(* Logix 5000 project; controller Amvex_Thorpe_Flowmeter vendor 1 type 14 code 106 rev 33.13; software revision 33.01; part 2 of 16 *)
(* tags used below, declared in another part *)
   Close : BOOL;
   Delay : TIMER;
   Open : BOOL;

ADD_ON_INSTRUCTION Banner_XS26_RCD_Function   (* revision 1.1, vendor Banner Engineering *)
// This AOI goes through a Virtual Reset or Cancel Delay request from the PLC to the XS26 Safety Controller.
VAR_IN_OUT
   RCD_Desired_Code : INT; {required}   // Numerical code that will be sent to the XS26 controller.
   RCD_Actuation_Code : INT; {required}   // Location of Actuation Code in the XS26 Controller.
   RCD_Actuation_Code_Feedback : INT; {required}   // When the Reset or Cancel Delay is successfull the Actuation Code is stored into this location.
   RCD_Bit : BOOL; {required}   // Bit that activates a singular Reset or Cancel Delay function.
   RCD_Bit_Feedback : BOOL; {required}   // Feedback bit from the XS26 controller for the RCD_Bit.
   Reset_Control_Bit : BOOL; {required}   // Bit that is turned off after the AOI completes.
   Routine_Error : BOOL; {required}
END_VAR
VAR
   Routine_Control_Bit : SINT; {access None}   // Controls operation of the AOI.
   Timer : TIMER := (PRE := 3000); {access None}
   Halt : DINT; {access None}
END_VAR

ROUTINE Logic   (* ladder *)
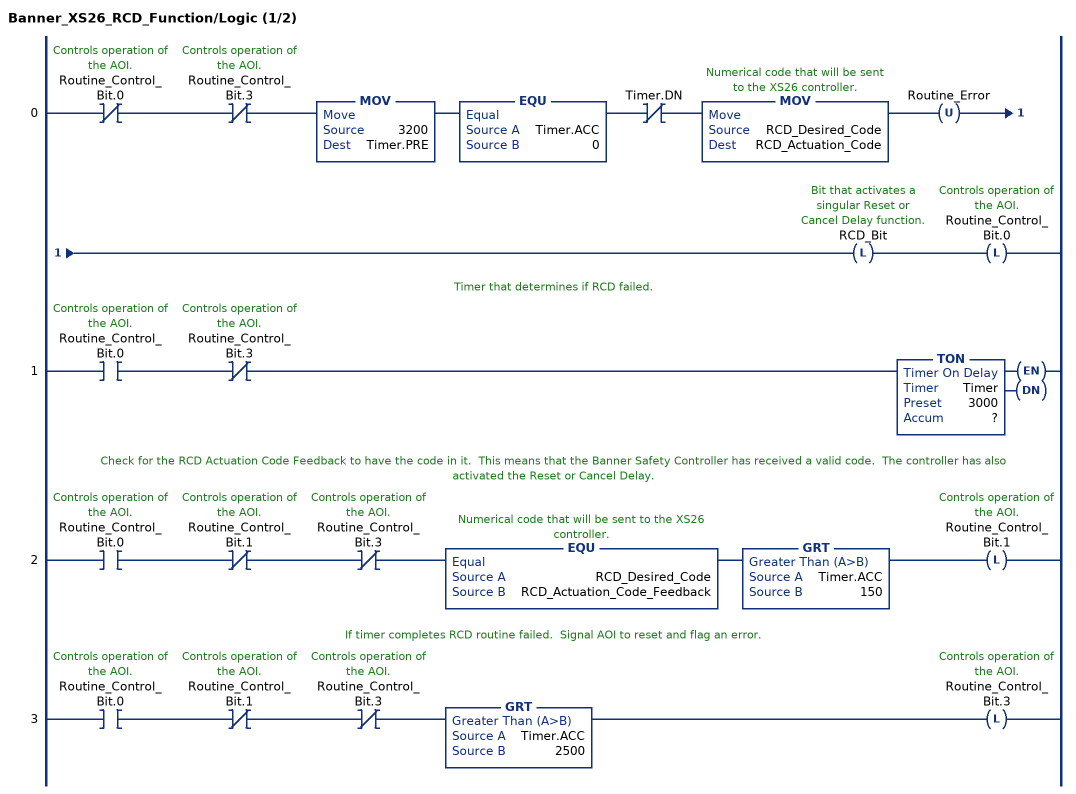
   0: XIO(Routine_Control_Bit.0)XIO(Routine_Control_Bit.3)MOV(3200,Timer.PRE)EQU(Timer.ACC,0)XIO(Timer.DN)MOV(RCD_Desired_Code,RCD_Actuation_Code)OTU(Routine_Error)OTL(RCD_Bit)OTL(Routine_Control_Bit.0);
   // Timer that determines if RCD failed.
   1: XIC(Routine_Control_Bit.0)XIO(Routine_Control_Bit.3)TON(Timer,?,?);
   // Check for the RCD Actuation Code Feedback to have the code in it.  This means that the Banner Safety Controller has received a valid code.  The controller has also activated the Reset or Cancel Delay.
   2: XIC(Routine_Control_Bit.0)XIO(Routine_Control_Bit.1)XIO(Routine_Control_Bit.3)EQU(RCD_Desired_Code,RCD_Actuation_Code_Feedback)GRT(Timer.ACC,150)OTL(Routine_Control_Bit.1);
   // If timer completes RCD routine failed.  Signal AOI to reset and flag an error.
   3: XIC(Routine_Control_Bit.0)XIO(Routine_Control_Bit.1)XIO(Routine_Control_Bit.3)GRT(Timer.ACC,2500)OTL(Routine_Control_Bit.3);
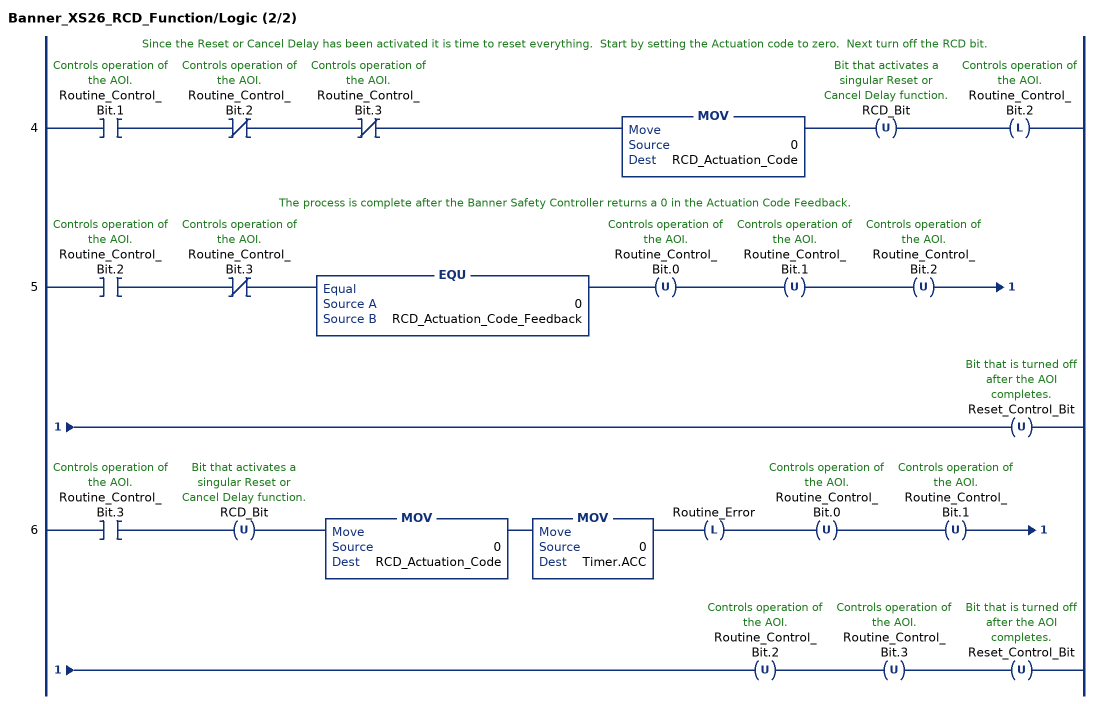
   // Since the Reset or Cancel Delay has been activated it is time to reset everything.  Start by setting the Actuation code to zero.  Next turn off the RCD bit.
   4: XIC(Routine_Control_Bit.1)XIO(Routine_Control_Bit.2)XIO(Routine_Control_Bit.3)MOV(0,RCD_Actuation_Code)OTU(RCD_Bit)OTL(Routine_Control_Bit.2);
   // The process is complete after the Banner Safety Controller returns a 0 in the Actuation Code Feedback.
   5: XIC(Routine_Control_Bit.2)XIO(Routine_Control_Bit.3)EQU(0,RCD_Actuation_Code_Feedback)OTU(Routine_Control_Bit.0)OTU(Routine_Control_Bit.1)OTU(Routine_Control_Bit.2)OTU(Reset_Control_Bit);
   6: XIC(Routine_Control_Bit.3)OTU(RCD_Bit)MOV(0,RCD_Actuation_Code)MOV(0,Timer.ACC)OTL(Routine_Error)OTU(Routine_Control_Bit.0)OTU(Routine_Control_Bit.1)OTU(Routine_Control_Bit.2)OTU(Routine_Control_Bit.3)OTU(Reset_Control_Bit);
END_ROUTINE
END_ADD_ON_INSTRUCTION

ADD_ON_INSTRUCTION Connect   (* revision 0.1, vendor Mecademic Inc. *)
// Monitor the robot module connection
VAR_IN_OUT
   RobotInstance : MODULE; {required}
END_VAR
VAR_INPUT
   Connect : BOOL; {access None, required}
END_VAR
VAR_OUTPUT
   RobotConnected : BOOL; {visible}
   ConnectionInhibited : BOOL; {visible}
   ConnectionFailed : BOOL; {visible}
END_VAR
VAR
   ConnectValue : DINT; {access None}
   DisconnectValue : DINT := 4; {access None}
   RobotInstance_Status : DINT; {access None}
   RobotInstance_Status_Masked : DINT; {access None}
END_VAR

ROUTINE Logic   (* ladder *)
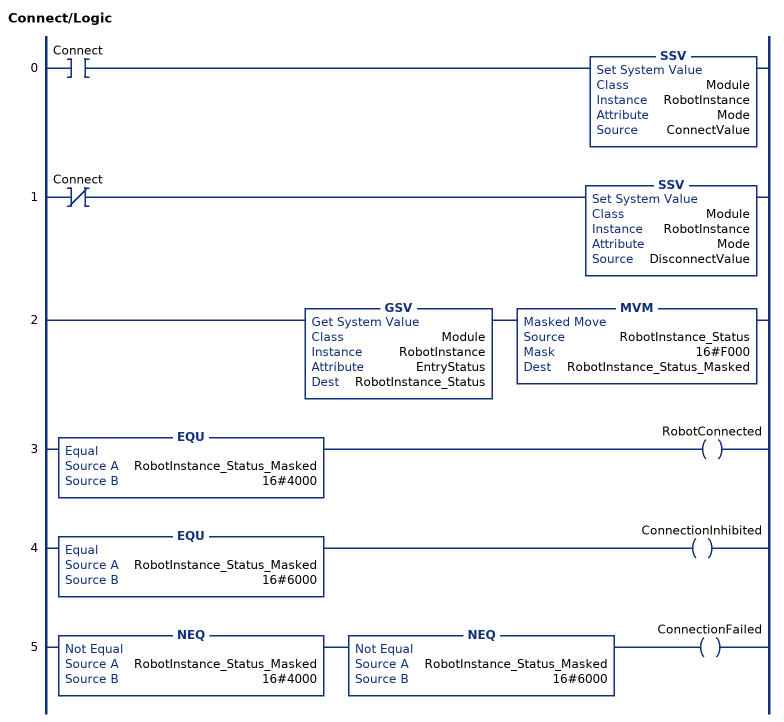
   0: XIC(Connect)SSV(Module,RobotInstance,Mode,ConnectValue);
   1: XIO(Connect)SSV(Module,RobotInstance,Mode,DisconnectValue);
   2: GSV(Module,RobotInstance,EntryStatus,RobotInstance_Status)MVM(RobotInstance_Status,16#F000,RobotInstance_Status_Masked);
   3: EQU(RobotInstance_Status_Masked,16#4000)OTE(RobotConnected);
   4: EQU(RobotInstance_Status_Masked,16#6000)OTE(ConnectionInhibited);
   5: NEQ(RobotInstance_Status_Masked,16#4000)NEQ(RobotInstance_Status_Masked,16#6000)OTE(ConnectionFailed);
END_ROUTINE
END_ADD_ON_INSTRUCTION

ADD_ON_INSTRUCTION Delay   (* revision 0.1, vendor Mecademic Inc., ExecuteEnableInFalse *)
// Delay in seconds before processing the next command
VAR_IN_OUT
   RobotInputs : _061D:Meca500_86BDA20B:I:0; {required}
   RobotOutputs : _061D:Meca500_01F88326:O:0; {required}
END_VAR
VAR_INPUT
   Parameter_Value : REAL; {required}
   ExternalStateControl : BOOL; {required}
   ExternalMoveID : INT; {required}
END_VAR
VAR_OUTPUT
   Enabled : BOOL; {visible}
   Sent : BOOL; {visible}
   Buffered : BOOL; {visible}
   Error : BOOL; {visible}
END_VAR
VAR
   InternalMoveID : INT; {access None}
   MoveIDTrig : BOOL; {access None}
   MoveIDUpdated : BOOL; {access None}
   OneShot : DINT; {access None}
   FirstScan : BOOL; {access None}
END_VAR

ROUTINE EnableInFalse   (* ladder *)
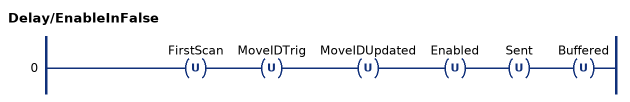
   0: OTU(FirstScan)OTU(MoveIDTrig)OTU(MoveIDUpdated)OTU(Enabled)OTU(Sent)OTU(Buffered);
END_ROUTINE

ROUTINE Logic   (* ladder *)
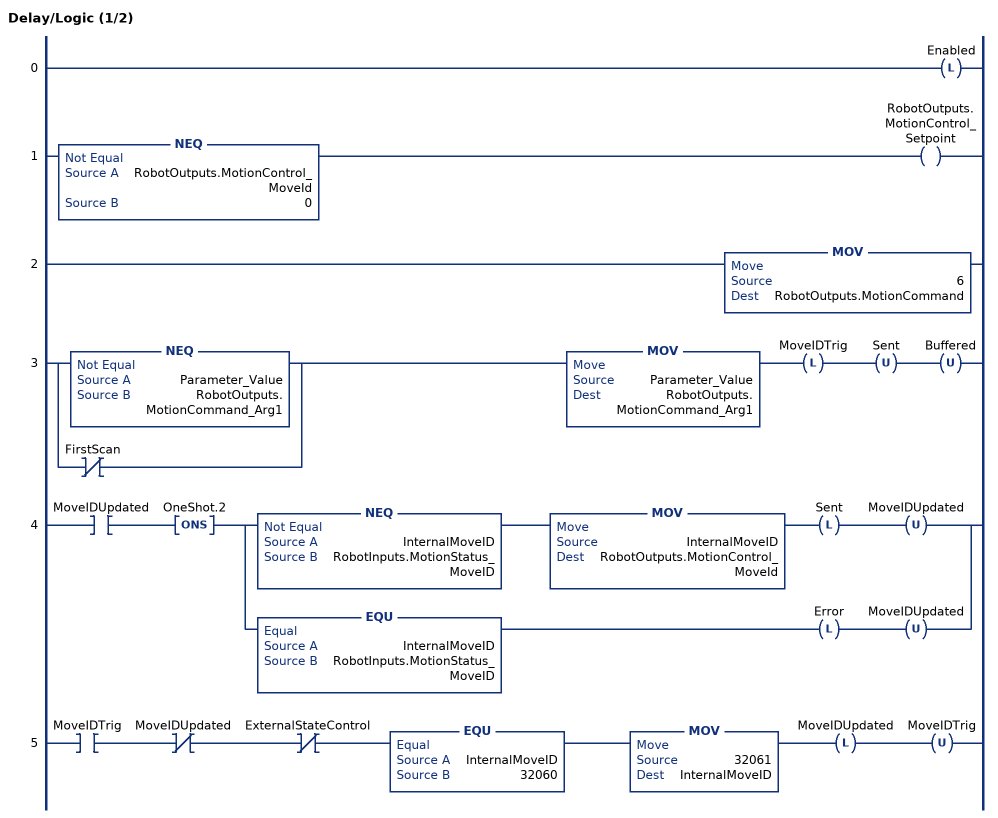
   0: OTL(Enabled);
   1: NEQ(RobotOutputs.MotionControl_MoveId,0)OTE(RobotOutputs.MotionControl_Setpoint);
   2: MOV(6,RobotOutputs.MotionCommand);
   3: [NEQ(Parameter_Value,RobotOutputs.MotionCommand_Arg1) ,XIO(FirstScan) ]MOV(Parameter_Value,RobotOutputs.MotionCommand_Arg1)OTL(MoveIDTrig)OTU(Sent)OTU(Buffered);
   4: XIC(MoveIDUpdated)ONS(OneShot.2)[NEQ(InternalMoveID,RobotInputs.MotionStatus_MoveID) MOV(InternalMoveID,RobotOutputs.MotionControl_MoveId) OTL(Sent) OTU(MoveIDUpdated) ,EQU(InternalMoveID,RobotInputs.MotionStatus_MoveID) OTL(Error) OTU(MoveIDUpdated) ];
   5: XIC(MoveIDTrig)XIO(MoveIDUpdated)XIO(ExternalStateControl)EQU(InternalMoveID,32060)MOV(32061,InternalMoveID)OTL(MoveIDUpdated)OTU(MoveIDTrig);
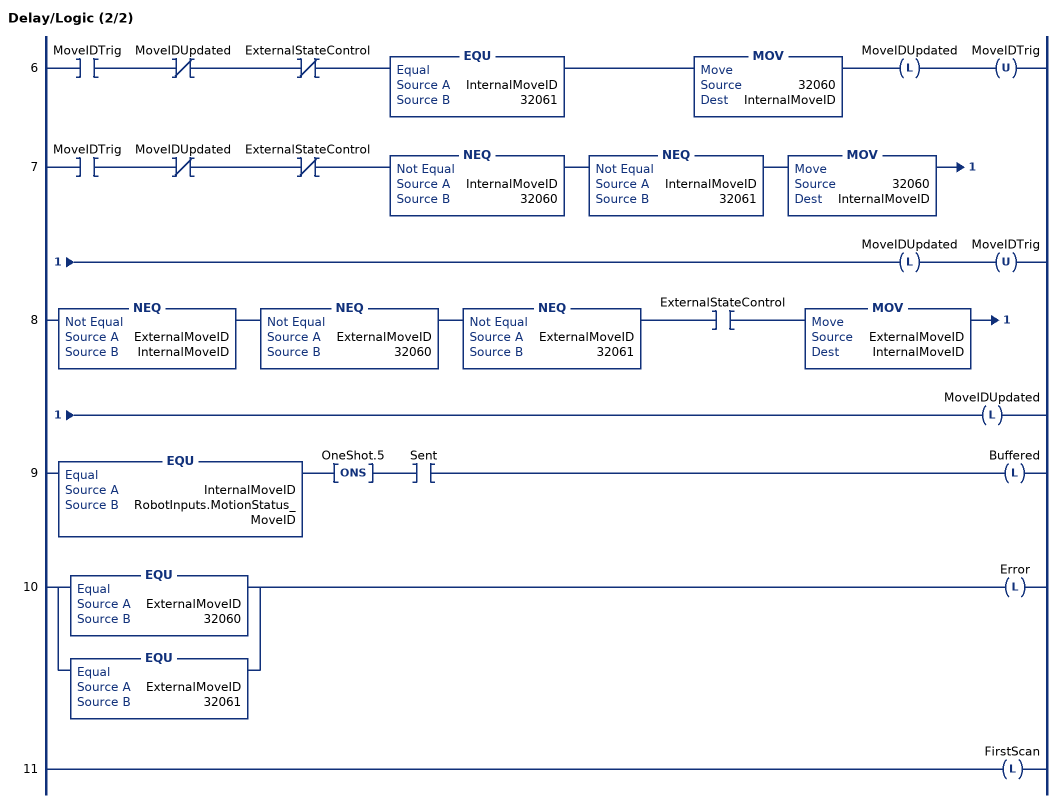
   6: XIC(MoveIDTrig)XIO(MoveIDUpdated)XIO(ExternalStateControl)EQU(InternalMoveID,32061)MOV(32060,InternalMoveID)OTL(MoveIDUpdated)OTU(MoveIDTrig);
   7: XIC(MoveIDTrig)XIO(MoveIDUpdated)XIO(ExternalStateControl)NEQ(InternalMoveID,32060)NEQ(InternalMoveID,32061)MOV(32060,InternalMoveID)OTL(MoveIDUpdated)OTU(MoveIDTrig);
   8: NEQ(ExternalMoveID,InternalMoveID)NEQ(ExternalMoveID,32060)NEQ(ExternalMoveID,32061)XIC(ExternalStateControl)MOV(ExternalMoveID,InternalMoveID)OTL(MoveIDUpdated);
   9: EQU(InternalMoveID,RobotInputs.MotionStatus_MoveID)ONS(OneShot.5)XIC(Sent)OTL(Buffered);
   10: [EQU(ExternalMoveID,32060) ,EQU(ExternalMoveID,32061) ]OTL(Error);
   11: OTL(FirstScan);
END_ROUTINE
END_ADD_ON_INSTRUCTION

ADD_ON_INSTRUCTION FAULT_AOI   (* revision 1.0, vendor Envision Automation & Controls *)
VAR_INPUT
   Fault : BOOL; {required}
   Bypass : BOOL; {required}
   Timer_PRE : DINT; {required}
END_VAR
VAR_OUTPUT
   Timer_ACC : DINT; {visible}
   Faulted : BOOL; {access Read Only, required}
END_VAR
VAR_INPUT
   Reset : BOOL; {access Read Only, required}
END_VAR
VAR
   Timer : TIMER; {access None}
END_VAR

ROUTINE Logic   (* ladder *)
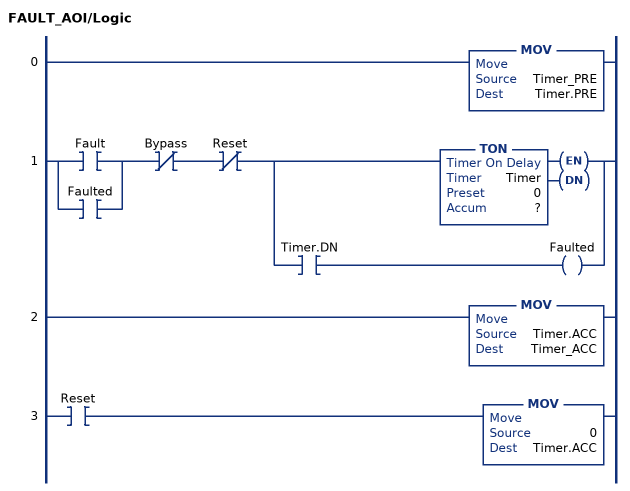
   0: MOV(Timer_PRE,Timer.PRE);
   1: [XIC(Fault) ,XIC(Faulted) ]XIO(Bypass)XIO(Reset)[TON(Timer,?,?) ,XIC(Timer.DN) OTE(Faulted) ];
   2: MOV(Timer.ACC,Timer_ACC);
   3: XIC(Reset)MOV(0,Timer.ACC);
END_ROUTINE
END_ADD_ON_INSTRUCTION

ADD_ON_INSTRUCTION GripperControl   (* revision 0.1, vendor Mecademic Inc., ExecuteEnableInFalse *)
// Open or close the gripper
VAR_IN_OUT
   RobotInputs : _061D:Meca500_86BDA20B:I:0; {required}
   RobotOutputs : _061D:Meca500_01F88326:O:0; {required}
END_VAR
VAR_INPUT
   Parameter_Value : REAL; {required}
   ExternalStateControl : BOOL; {required}
   ExternalMoveID : INT; {required}
END_VAR
VAR_OUTPUT
   Enabled : BOOL; {visible}
   Sent : BOOL; {visible}
   Buffered : BOOL; {visible}
   Error : BOOL; {visible}
END_VAR
VAR
   InternalMoveID : INT; {access None}
   MoveIDTrig : BOOL; {access None}
   MoveIDUpdated : BOOL; {access None}
   OneShot : DINT; {access None}
   FirstScan : BOOL; {access None}
END_VAR

ROUTINE EnableInFalse   (* ladder *)
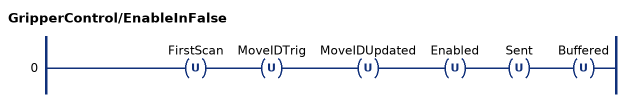
   0: OTU(FirstScan)OTU(MoveIDTrig)OTU(MoveIDUpdated)OTU(Enabled)OTU(Sent)OTU(Buffered);
END_ROUTINE

ROUTINE Logic   (* ladder *)
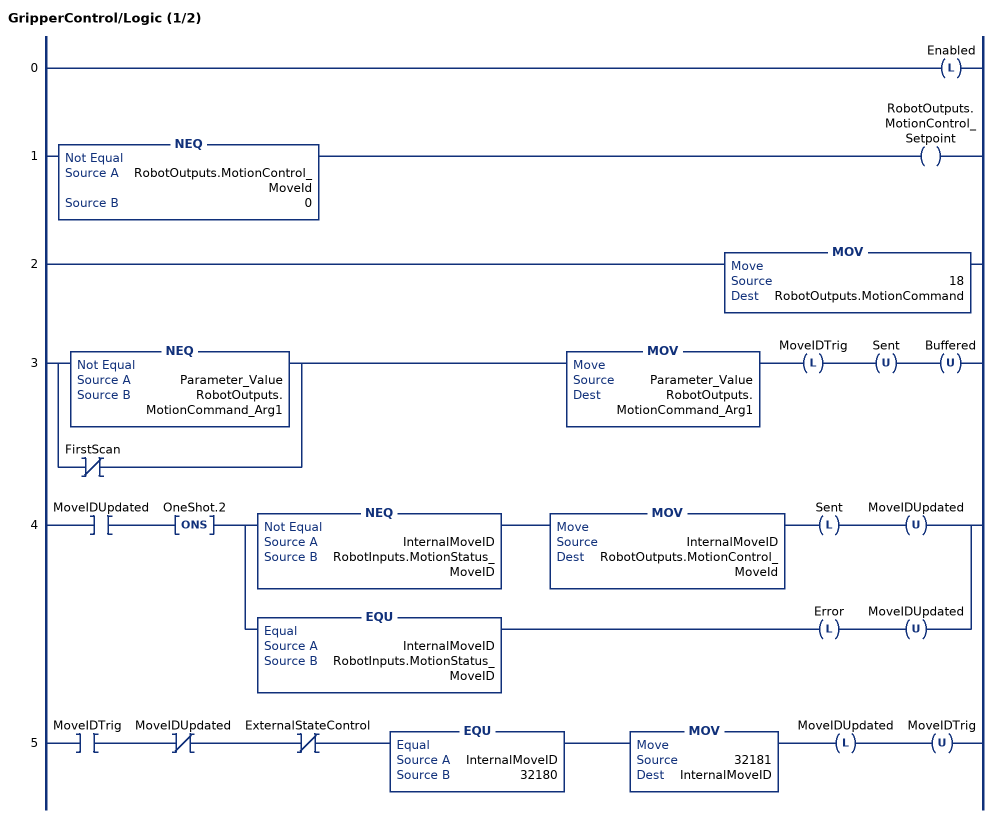
   0: OTL(Enabled);
   1: NEQ(RobotOutputs.MotionControl_MoveId,0)OTE(RobotOutputs.MotionControl_Setpoint);
   2: MOV(18,RobotOutputs.MotionCommand);
   3: [NEQ(Parameter_Value,RobotOutputs.MotionCommand_Arg1) ,XIO(FirstScan) ]MOV(Parameter_Value,RobotOutputs.MotionCommand_Arg1)OTL(MoveIDTrig)OTU(Sent)OTU(Buffered);
   4: XIC(MoveIDUpdated)ONS(OneShot.2)[NEQ(InternalMoveID,RobotInputs.MotionStatus_MoveID) MOV(InternalMoveID,RobotOutputs.MotionControl_MoveId) OTL(Sent) OTU(MoveIDUpdated) ,EQU(InternalMoveID,RobotInputs.MotionStatus_MoveID) OTL(Error) OTU(MoveIDUpdated) ];
   5: XIC(MoveIDTrig)XIO(MoveIDUpdated)XIO(ExternalStateControl)EQU(InternalMoveID,32180)MOV(32181,InternalMoveID)OTL(MoveIDUpdated)OTU(MoveIDTrig);
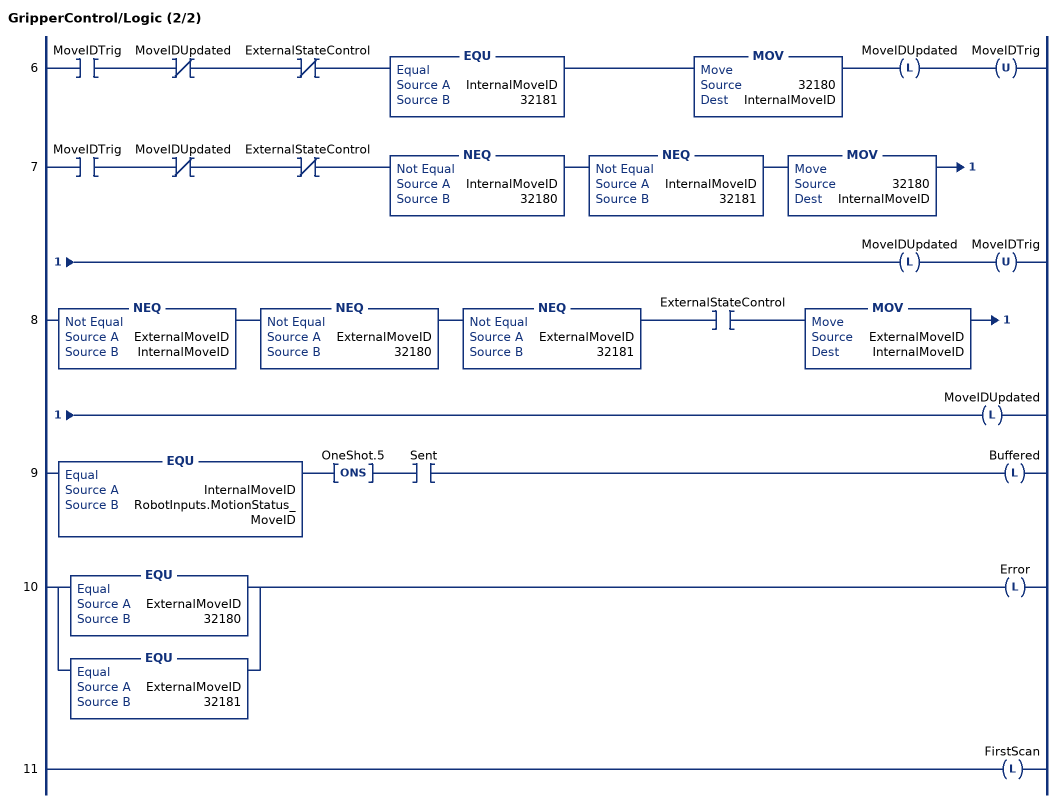
   6: XIC(MoveIDTrig)XIO(MoveIDUpdated)XIO(ExternalStateControl)EQU(InternalMoveID,32181)MOV(32180,InternalMoveID)OTL(MoveIDUpdated)OTU(MoveIDTrig);
   7: XIC(MoveIDTrig)XIO(MoveIDUpdated)XIO(ExternalStateControl)NEQ(InternalMoveID,32180)NEQ(InternalMoveID,32181)MOV(32180,InternalMoveID)OTL(MoveIDUpdated)OTU(MoveIDTrig);
   8: NEQ(ExternalMoveID,InternalMoveID)NEQ(ExternalMoveID,32180)NEQ(ExternalMoveID,32181)XIC(ExternalStateControl)MOV(ExternalMoveID,InternalMoveID)OTL(MoveIDUpdated);
   9: EQU(InternalMoveID,RobotInputs.MotionStatus_MoveID)ONS(OneShot.5)XIC(Sent)OTL(Buffered);
   10: [EQU(ExternalMoveID,32180) ,EQU(ExternalMoveID,32181) ]OTL(Error);
   11: OTL(FirstScan);
END_ROUTINE
END_ADD_ON_INSTRUCTION

ADD_ON_INSTRUCTION GripperPos   (* revision 1.0, vendor Mecademic.inc, ExecuteEnableInFalse *)
// Move Gripper to a specific position, in mm from the most closed position
VAR_IN_OUT
   RobotOutputs : _061D:Meca500_01F88326:O:0; {required}
   RobotInputs : _061D:Meca500_86BDA20B:I:0; {required}
END_VAR
VAR_INPUT
   Parameter_Value : DINT; {access None, required}
   ExternalStateControl : BOOL; {required}
   ExternalMoveID : DINT; {required}
END_VAR
VAR_OUTPUT
   Enabled : BOOL; {visible}
   Sent : BOOL; {access Read Only, visible}
   Buffered : BOOL; {access Read Only, visible}
   Error : BOOL; {access Read Only, visible}
END_VAR
VAR
   MoveIDTrig : BOOL; {access None}
   MoveIDUpdated : BOOL; {access None}
   OneShot : DINT; {access None}
   InternalMoveID : DINT; {access None}
   FirstScan : BOOL; {access None}
END_VAR

ROUTINE EnableInFalse   (* ladder *)
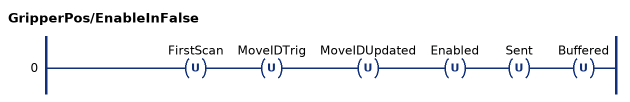
   0: OTU(FirstScan)OTU(MoveIDTrig)OTU(MoveIDUpdated)OTU(Enabled)OTU(Sent)OTU(Buffered);
END_ROUTINE

ROUTINE Logic   (* ladder *)
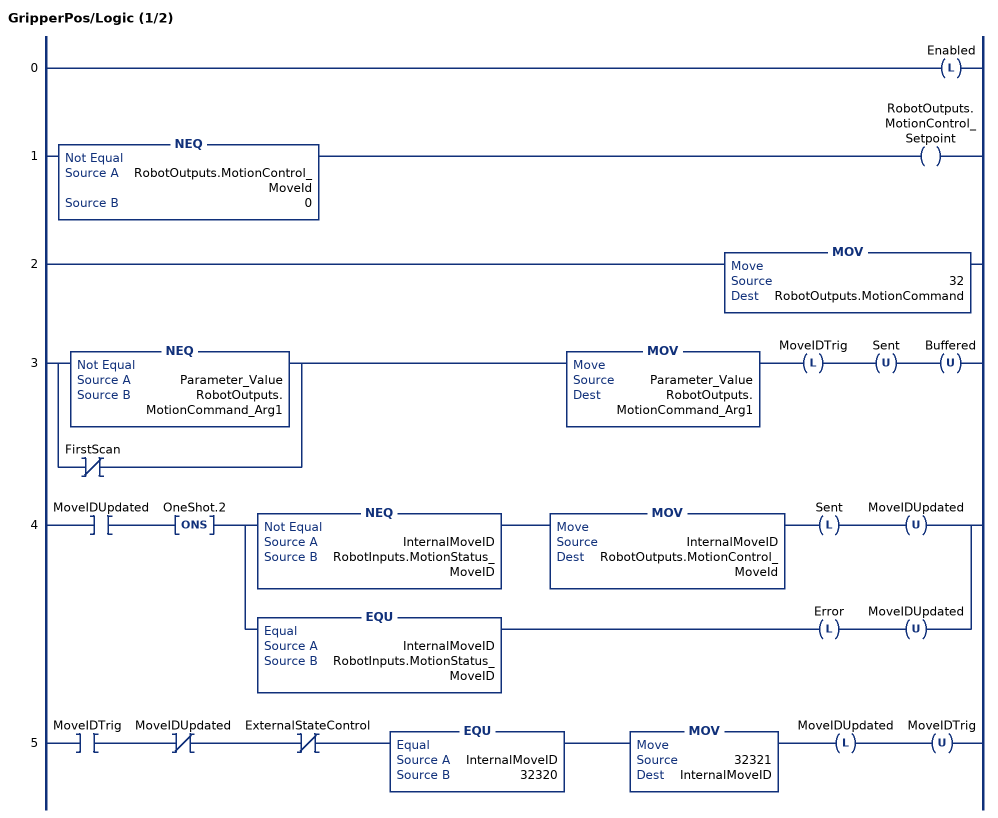
   0: OTL(Enabled);
   1: NEQ(RobotOutputs.MotionControl_MoveId,0)OTE(RobotOutputs.MotionControl_Setpoint);
   2: MOV(32,RobotOutputs.MotionCommand);
   3: [NEQ(Parameter_Value,RobotOutputs.MotionCommand_Arg1) ,XIO(FirstScan) ]MOV(Parameter_Value,RobotOutputs.MotionCommand_Arg1)OTL(MoveIDTrig)OTU(Sent)OTU(Buffered);
   4: XIC(MoveIDUpdated)ONS(OneShot.2)[NEQ(InternalMoveID,RobotInputs.MotionStatus_MoveID) MOV(InternalMoveID,RobotOutputs.MotionControl_MoveId) OTL(Sent) OTU(MoveIDUpdated) ,EQU(InternalMoveID,RobotInputs.MotionStatus_MoveID) OTL(Error) OTU(MoveIDUpdated) ];
   5: XIC(MoveIDTrig)XIO(MoveIDUpdated)XIO(ExternalStateControl)EQU(InternalMoveID,32320)MOV(32321,InternalMoveID)OTL(MoveIDUpdated)OTU(MoveIDTrig);
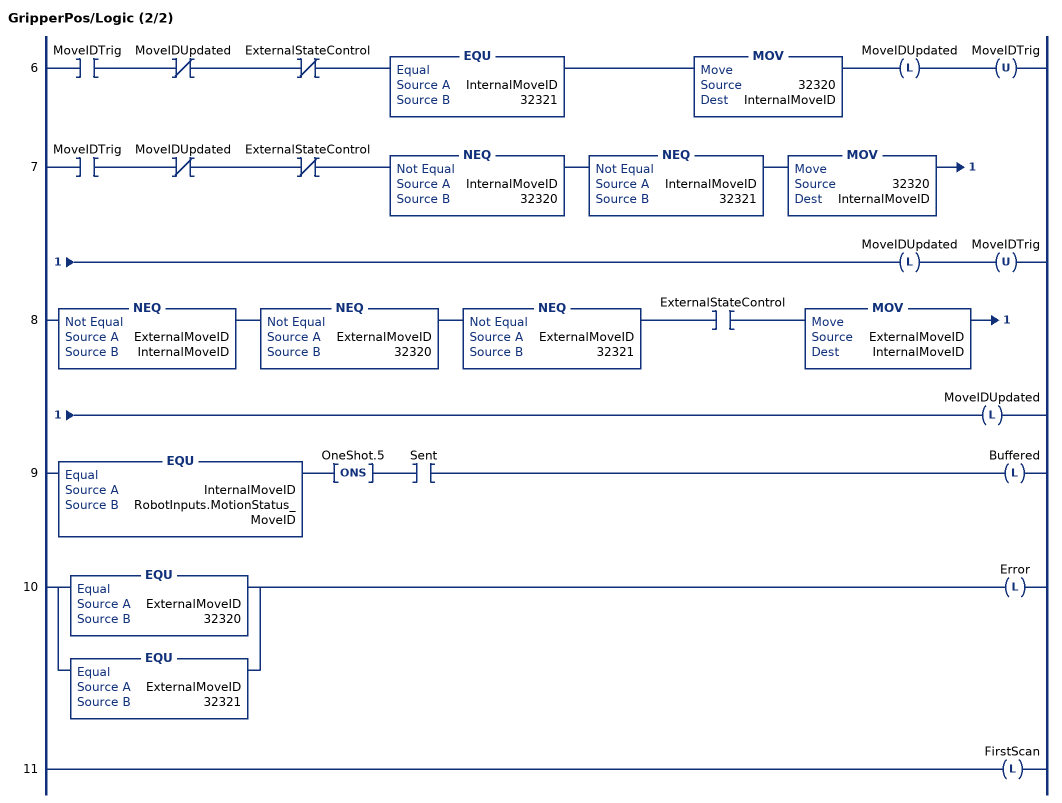
   6: XIC(MoveIDTrig)XIO(MoveIDUpdated)XIO(ExternalStateControl)EQU(InternalMoveID,32321)MOV(32320,InternalMoveID)OTL(MoveIDUpdated)OTU(MoveIDTrig);
   7: XIC(MoveIDTrig)XIO(MoveIDUpdated)XIO(ExternalStateControl)NEQ(InternalMoveID,32320)NEQ(InternalMoveID,32321)MOV(32320,InternalMoveID)OTL(MoveIDUpdated)OTU(MoveIDTrig);
   8: NEQ(ExternalMoveID,InternalMoveID)NEQ(ExternalMoveID,32320)NEQ(ExternalMoveID,32321)XIC(ExternalStateControl)MOV(ExternalMoveID,InternalMoveID)OTL(MoveIDUpdated);
   9: EQU(InternalMoveID,RobotInputs.MotionStatus_MoveID)ONS(OneShot.5)XIC(Sent)OTL(Buffered);
   10: [EQU(ExternalMoveID,32320) ,EQU(ExternalMoveID,32321) ]OTL(Error);
   11: OTL(FirstScan);
END_ROUTINE
END_ADD_ON_INSTRUCTION

ADD_ON_INSTRUCTION GripperRange   (* revision 1.0, vendor Mecademic inc., ExecuteEnableInFalse *)
// Set the Close and Open position that will be used when calling GripperClose and GripperOpen
VAR_IN_OUT
   RobotOutputs : _061D:Meca500_01F88326:O:0; {required}
   RobotInputs : _061D:Meca500_86BDA20B:I:0; {required}
END_VAR
VAR_INPUT
   Closed_Position : REAL; {required}   // in mm
   Opened_Position : REAL; {required}   // in mm
   ExternalStateControl : BOOL; {required}
   ExternalMoveID : INT; {required}
END_VAR
VAR_OUTPUT
   Enabled : BOOL; {access Read Only, visible}
   Sent : BOOL; {access Read Only, visible}
   Buffered : BOOL; {access Read Only, visible}
   Error : BOOL; {access Read Only, visible}
END_VAR
VAR
   MoveIDTrig : BOOL; {access None}
   FirstScan : BOOL; {access None}
   MoveIDUpdated : BOOL; {access None}
   OneShot : DINT; {access None}
   InternalMoveID : INT; {access None}
END_VAR

ROUTINE EnableInFalse   (* ladder *)
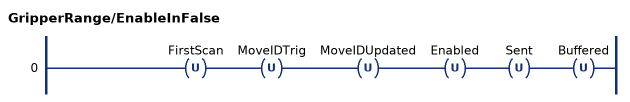
   0: OTU(FirstScan)OTU(MoveIDTrig)OTU(MoveIDUpdated)OTU(Enabled)OTU(Sent)OTU(Buffered);
END_ROUTINE

ROUTINE Logic   (* ladder *)
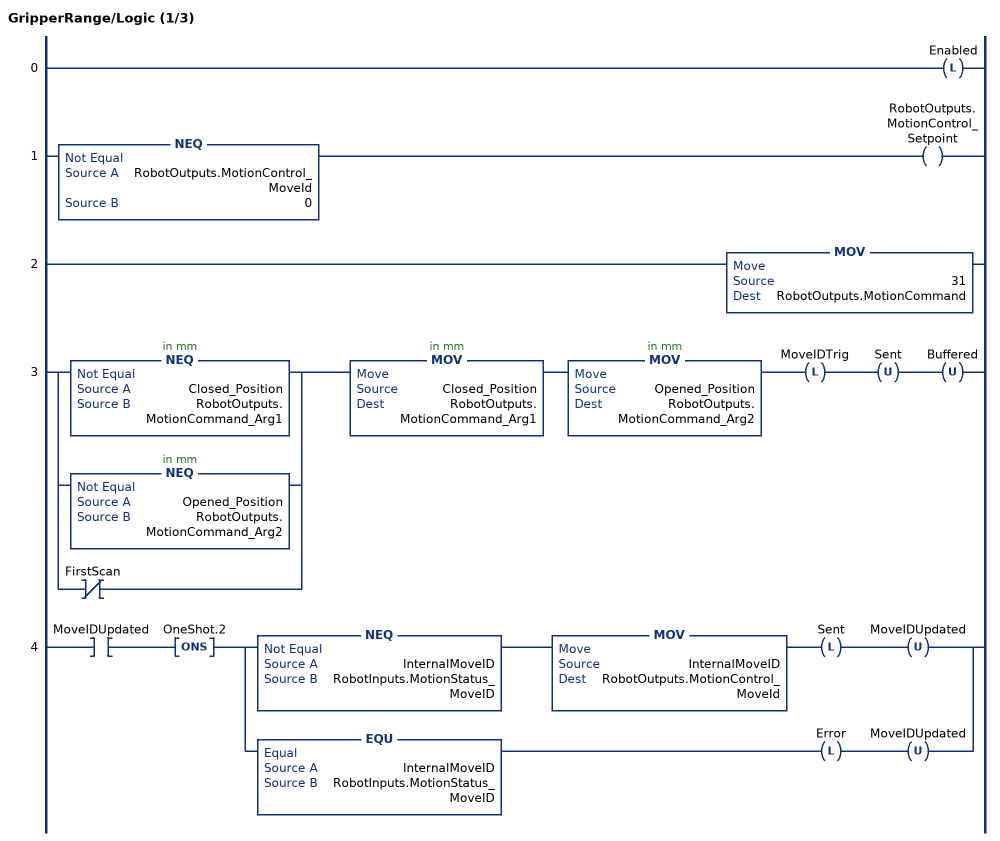
   0: OTL(Enabled);
   1: NEQ(RobotOutputs.MotionControl_MoveId,0)OTE(RobotOutputs.MotionControl_Setpoint);
   2: MOV(31,RobotOutputs.MotionCommand);
   3: [NEQ(Closed_Position,RobotOutputs.MotionCommand_Arg1) ,NEQ(Opened_Position,RobotOutputs.MotionCommand_Arg2) ,XIO(FirstScan) ]MOV(Closed_Position,RobotOutputs.MotionCommand_Arg1)MOV(Opened_Position,RobotOutputs.MotionCommand_Arg2)OTL(MoveIDTrig)OTU(Sent)OTU(Buffered);
   4: XIC(MoveIDUpdated)ONS(OneShot.2)[NEQ(InternalMoveID,RobotInputs.MotionStatus_MoveID) MOV(InternalMoveID,RobotOutputs.MotionControl_MoveId) OTL(Sent) OTU(MoveIDUpdated) ,EQU(InternalMoveID,RobotInputs.MotionStatus_MoveID) OTL(Error) OTU(MoveIDUpdated) ];
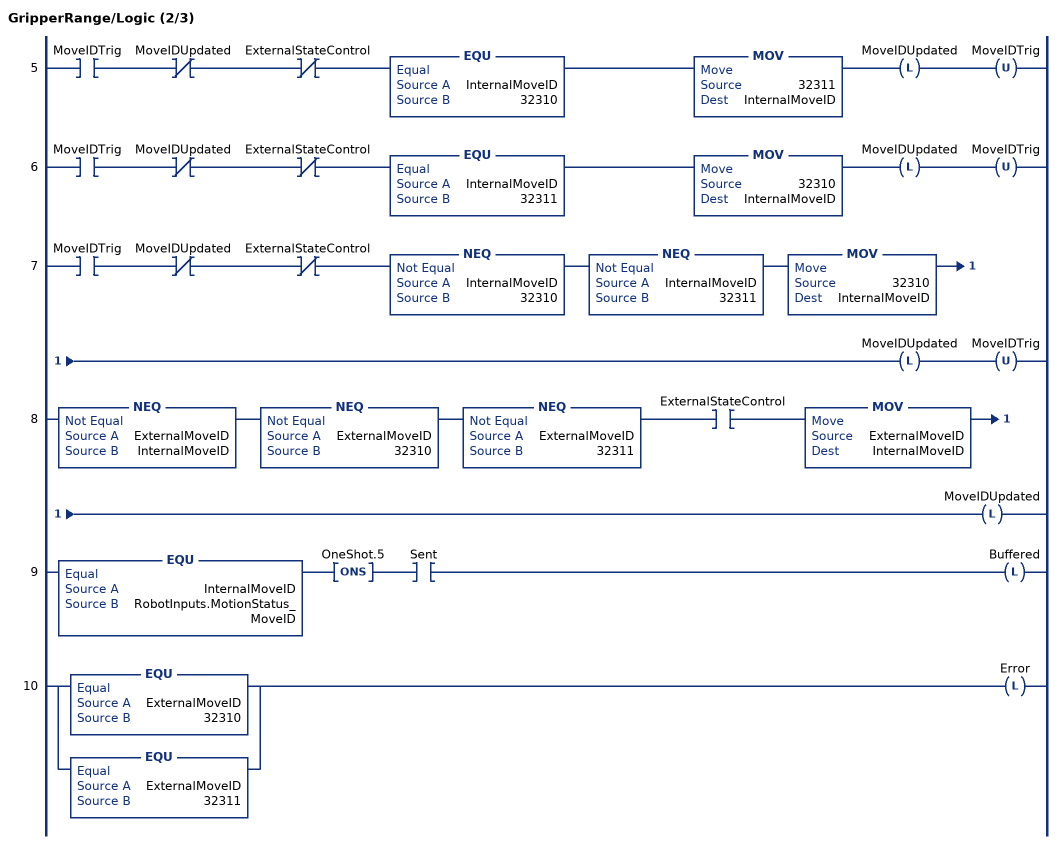
   5: XIC(MoveIDTrig)XIO(MoveIDUpdated)XIO(ExternalStateControl)EQU(InternalMoveID,32310)MOV(32311,InternalMoveID)OTL(MoveIDUpdated)OTU(MoveIDTrig);
   6: XIC(MoveIDTrig)XIO(MoveIDUpdated)XIO(ExternalStateControl)EQU(InternalMoveID,32311)MOV(32310,InternalMoveID)OTL(MoveIDUpdated)OTU(MoveIDTrig);
   7: XIC(MoveIDTrig)XIO(MoveIDUpdated)XIO(ExternalStateControl)NEQ(InternalMoveID,32310)NEQ(InternalMoveID,32311)MOV(32310,InternalMoveID)OTL(MoveIDUpdated)OTU(MoveIDTrig);
   8: NEQ(ExternalMoveID,InternalMoveID)NEQ(ExternalMoveID,32310)NEQ(ExternalMoveID,32311)XIC(ExternalStateControl)MOV(ExternalMoveID,InternalMoveID)OTL(MoveIDUpdated);
   9: EQU(InternalMoveID,RobotInputs.MotionStatus_MoveID)ONS(OneShot.5)XIC(Sent)OTL(Buffered);
   10: [EQU(ExternalMoveID,32310) ,EQU(ExternalMoveID,32311) ]OTL(Error);
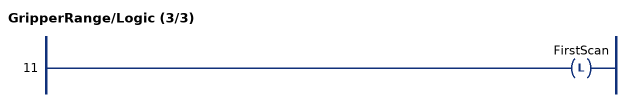
   11: OTL(FirstScan);
END_ROUTINE
END_ADD_ON_INSTRUCTION

ADD_ON_INSTRUCTION IvSwichPrgoram   (* revision 1.0, vendor KEYENCE CORPORATION *)
// AOI of Keyence IV for switching program
VAR_IN_OUT
   InModuleData : INT[197]; {required}
   OutModuleData : INT[6]; {required}
END_VAR
VAR_INPUT
   SwitchProgramRequest : BOOL; {access None}
   TargetProgramNo : INT;
END_VAR
VAR_OUTPUT
   SwitchProgramDone : BOOL; {access Read Only}
END_VAR
VAR
   ONS : BOOL[32]; {access None}
   DoneCheckForSwitchProgram : BOOL; {access None}
END_VAR

ROUTINE Logic   (* ladder *)
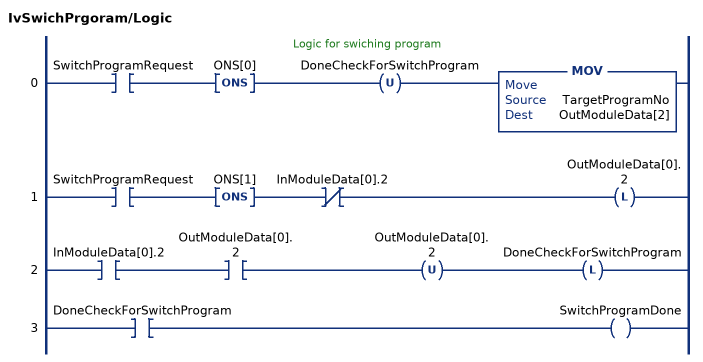
   // Logic for swiching program
   0: XIC(SwitchProgramRequest)ONS(ONS[0])OTU(DoneCheckForSwitchProgram)MOV(TargetProgramNo,OutModuleData[2]);
   1: XIC(SwitchProgramRequest)ONS(ONS[1])XIO(InModuleData[0].2)OTL(OutModuleData[0].2);
   2: XIC(InModuleData[0].2)XIC(OutModuleData[0].2)OTU(OutModuleData[0].2)OTL(DoneCheckForSwitchProgram);
   3: XIC(DoneCheckForSwitchProgram)OTE(SwitchProgramDone);
END_ROUTINE
END_ADD_ON_INSTRUCTION
